Yaskawa INFORM job: START-ML.JBI

/JOB
//NAME START-ML
///FOLDERNAME FOLDER001
//POS
///NPOS 0,0,0,0,0,0
//INST
///DATE 2025/09/30 17:15
///ATTR SC,RW
///GROUP1 RB1
NOP
SET B096 10
SET B097 0
SET B098 0
SET B099 0
CALL JOB:MULTI-ABOVE ARGF1
CALL JOB:ABOVE-TO-BELOW
CALL JOB:MULTI-BELOW ARGF3
CALL JOB:BELOW-TO-ABOVE
CALL JOB:MULTI-ABOVE ARGF2
CALL JOB:ABOVE-TO-BELOW
CALL JOB:MULTI-BELOW ARGF2
CALL JOB:BELOW-TO-ABOVE
CALL JOB:MULTI-ABOVE ARGF2
CALL JOB:ABOVE-TO-BELOW
CALL JOB:MULTI-BELOW ARGF3
CALL JOB:BELOW-TO-ABOVE
CALL JOB:MULTI-ABOVE ARGF3
CALL JOB:ABOVE-TO-BELOW
CALL JOB:MULTI-BELOW ARGF4
CALL JOB:BELOW-TO-ABOVE
CALL JOB:MULTI-ABOVE ARGF4
CALL JOB:ABOVE-TO-BELOW
CALL JOB:MULTI-BELOW ARGF5
CALL JOB:BELOW-TO-ABOVE
CALL JOB:MULTI-ABOVE ARGF5
CALL JOB:GO-START
CALL JOB:GO-PARK
END
